(* PLC project Generated.project, CODESYS CODESYS V3.5 SP19 Patch 1 *)
(* stored: creationDateTime 2026-09-03T14:40:30.920452, modificationDateTime 2026-09-03T14:40:30.920452 *)

(* ═══════════════════════════════════════════════════════════════ ⚙️ ST_MachineHomingCfg — Réglages IHM du cycle de référencement machine ─────────────────────────────────────────────────────────────── 🎯 Mise en service. Les réglages géométriques (positions capteur, offsets benne) restent portés par GVL_PERSISTENT (_WinchM1CfgPersist / _BucketCfgPersist). 💾 Ponté vers persist (_MachineHomingCfgPersist) via FB_CfgPersistBridge_MachineHomingCfg. ═══════════════════════════════════════════════════════════════ *)
TYPE ST_MachineHomingCfg : STRUCT
  ForceStepTarget : INT := 0;  (* 🔧 Step GRAFCET cible du forçage (0=HX0 .. 9=HXF), borné côté FB *)
  Initialized : BOOL := FALSE;  (* 🚦 flag restauration boot *)
END_STRUCT;
END_TYPE

(* ======================================================================= 💾 FB_CfgPersistBridge_MachineHomingCfg — Pont persistance pour ST_MachineHomingCfg ─────────────────────────────────────────────────────────────── 🎯 Rôle : Restauration et synchronisation bidirectionnelle IHM / Persist 💾 Persistance : Transfert GVL_PERSISTENT <-> GVL_IHM sur Initialized 📄 Doc métier : DOC/AF/AF_Partie-03_Contrats_Composants_v2.3.md §3 ======================================================================= *)
FUNCTION_BLOCK FB_CfgPersistBridge_MachineHomingCfg
  VAR_OUTPUT
    JustRestored : BOOL;  (* === ETATS RESTAURATION === <-- [STAT] Vrai sur le cycle de restauration initiale *)
  END_VAR
  VAR_IN_OUT
    Hmi : ST_MachineHomingCfg;  (* === BUS CONFIGURATION ET PERSISTANCE === <-> [BUS] Structure de configuration IHM *)
    Persist : ST_MachineHomingCfg;  (* <-> [BUS] Structure de configuration persistante *)
  END_VAR

            

JustRestored := FALSE;
IF NOT Hmi.Initialized THEN
    Hmi := Persist;
    Hmi.Initialized := TRUE;
    JustRestored := TRUE;
ELSE
    Persist := Hmi;
END_IF;

          
END_FUNCTION_BLOCK
